// A function block containing multiple file handling methods. 
// Note that the body of this FB does NOT need to be called as it holds no logic.
// All the methods should be called untill they return true, if they provide error information, 
// it will be trough a reference variable.
//
// For examples refer to tests in the folder "TESTS/Test suites", file "FB_FileHandlerTests".

{attribute 'no_explicit_call' := 'Body contains no logic, calling methods only allowed.'}
FUNCTION_BLOCK FB_FileHandler EXTENDS ZigaLibs_Core.FB_ErrorSource IMPLEMENTS I_FileHandler

VAR
	_fileInfo		: ST_FileInfo;
	_netId			: Tc2_System.T_AmsNetID;
	_lastOpenMode	: E_FileOpenMode;
	_streamEmpty	: BOOL := TRUE;
END_VAR

// Closes the file and returns TRUE when done.
METHOD Close : BOOL
Close := THIS^.CloseSilent(FALSE);
END_METHOD

// Closes the file without clearing the file properties.
METHOD PRIVATE CloseSilent : BOOL
VAR_INPUT
	silent	: BOOL; // IF set to TRUE, the file property won't be modified. To be used when flushing the stream.
END_VAR
VAR_INST
	fbFileClose	: Tc2_System.FB_FileClose;
END_VAR

VAR
	varInfo	: ZigaLibs_Core.T_VarInfo;
END_VAR
fbFileClose(
	bExecute := NOT fbFileClose.bBusy,
	hFile := File.Handle,
	sNetId := File.NetId);

IF NOT fbFileClose.bBusy THEN
	CloseSilent := TRUE;
	IF fbFileClose.bError THEN
		varInfo := __VARINFO(fbFileClose);
		THIS^.RaiseAdsError(Tc2_Standard.CONCAT(THIS^.InstancePath, varInfo.Symbol), fbFileClose.nErrId);
		THIS^.GenericError.Message := Tc2_Standard.CONCAT('An error occured when closing the file ', File.Name);
		fbFileClose(bExecute := FALSE);	
		RETURN;
	END_IF
	
	_streamEmpty := TRUE;
	fbFileClose(bExecute := FALSE);
	File.Handle := 0;	
	IF NOT silent THEN
		File.IsOpened := FALSE;
	END_IF
END_IF
END_METHOD

// Creates the file, if it does not yet exist,
METHOD Create : BOOL
VAR_INPUT
	path	: Tc2_System.T_MaxString;	// Path to the file location
	name	: Tc2_System.T_MaxString;	// Name of the file
	netId	: Tc2_System.T_AmsNetID;	// NetId where the file is located
END_VAR
VAR
	sb	: ZigaLibs_Core.FB_StringBuilder;
END_VAR
IF NOT file.IsOpened THEN
	THIS^.Open(
		path := path,
		name := name,
		mode := E_FileOpenMode.BINARY_APPEND_OVERWRITE_EXISTING,
		netId := netId);
		
	// Error opening the file, report and stop.
	IF THIS^.Error THEN
		THIS^.GenericError.Source := sb.Reset()
			.AddString(THIS^.InstancePath)
			.AddString('.Create()')
			.Create();
		
		THIS^.GenericError.Message := sb.Reset()
			.AddString('An error occurred when creating the file, while opening it:')
			.AddString(' Path = ').AddWithDblQuotationMarks(path)
			.AddString(' Name = ').AddWithDblQuotationMarks(name)
			.AddString(' NetId = ').AddWithDblQuotationMarks(netId)
			.AddString('. Refer to AdsError for more info.')
			.Create();
		Create := TRUE;
		RETURN;
	END_IF
ELSE
	Create := THIS^.Close();
	
	// Error closing the file. Report and stop.
	IF THIS^.Error THEN
		THIS^.GenericError.Source := sb.Reset()
			.AddString(THIS^.InstancePath)
			.AddString('.Create()')
			.Create();
		THIS^.GenericError.Message := sb.Reset()
			.AddString('An error occurred when creating the file, while closing it:')
			.AddString(' Path = ').AddWithDblQuotationMarks(path)
			.AddString(' Name = ').AddWithDblQuotationMarks(name)
			.AddString(' NetId = ').AddWithDblQuotationMarks(netId)
			.AddString('. Refer to AdsError for more info.')
			.Create();
	END_IF
END_IF
END_METHOD

{attribute 'monitoring':='call'}
(* Gets the current file properties.*)
PROPERTY File : REFERENCE TO ST_FileInfo
GET
File REF= _fileInfo;
END_GET
SET // PROTECTED
_fileInfo := File;
END_SET
END_PROPERTY

// Flushes the current file stream data to the file. 
// Basically file is closed and re-opened, which in turn writes the content of the stream to the file.
// If the file was opened to overwrite existing content, flushing will clear the data in the file!
// While flushing is being executed, the .File property DOES NOT CHANGE 
// For example, the File.IsOpened will remain TRUE even at the point where it is actually not. It will then be re-opened. 
// If an error occurs however, properties will be set to correct state.

METHOD Flush : BOOL
VAR_INST
	closeDone		: BOOL;
END_VAR
IF closeDone OR_ELSE THIS^.CloseSilent(TRUE) THEN
	// Error closing the file while flushing...
	IF THIS^.Error AND NOT closeDone THEN
		Flush := TRUE;
		THIS^.GenericError.Message := 'An error occurred while flushing the file stream (closing the file)...';
		THIS^.GenericError.Source := Tc2_Standard.CONCAT(THIS^.InstanceName, '.Flush()');
		RETURN;
	END_IF
	
	closeDone := TRUE;
END_IF

IF closeDone AND_THEN THIS^.Open(File.Path, File.Name, _lastOpenMode, File.NetId) THEN
	closeDone := FALSE;
	Flush := TRUE;
	// Error while opening the file while flushing...
	IF THIS^.Error THEN
		THIS^.File.Handle := 0;
		THIS^.File.IsOpened := FALSE;
		THIS^.GenericError.Message := 'An error occurred while flushing the file stream (opening the file)...';
		THIS^.GenericError.Source := Tc2_Standard.CONCAT(THIS^.InstanceName, '.Flush()');
	END_IF
END_IF
END_METHOD

// Opens the file in the path provided. If a file is already opened nothing happens.
// Returns: TRUE when done.
METHOD Open : BOOL
VAR_INPUT
	path	: Tc2_System.T_MaxString;	// Path to the file location
	name	: Tc2_System.T_MaxString;	// Name of the file
	mode	: E_FileOpenMode;			// Mode in which the file will be opened
	netId	: Tc2_System.T_AmsNetID;	// NetId where the file is located
END_VAR

VAR_INST
	fbFileOpen	: Tc2_System.FB_FileOpen;
END_VAR

VAR
	varInfo	: ZigaLibs_Core.T_VarInfo;
END_VAR
IF THIS^.File.Handle <> 0 THEN
	Open := TRUE;
	RETURN;
END_IF

fbFileOpen(
	bExecute := NOT fbFileOpen.bBusy,
	nMode := mode,
	sNetId := netID,
	sPathName := Utilities.Path.Generate().Join(path).Join(name).Create());
	
IF NOT fbFileOpen.bBusy THEN
	Open := TRUE;
	IF fbFileOpen.bError THEN
		varInfo := __VARINFO(fbFileOpen);
		THIS^.RaiseAdsError(Tc2_Standard.CONCAT(THIS^.InstancePath, varInfo.Symbol), fbFileOpen.nErrId);
		fbFileOpen(bExecute := FALSE);
		RETURN;
	END_IF
	_lastOpenMode := mode;
	fbFileOpen(bExecute := FALSE);
	File.Handle := fbFileOpen.hFile;
	File.Name := name;
	File.Path := path;
	File.NetId := netId;
	File.IsOpened := TRUE;
END_IF
END_METHOD

// Raise an error for a certain FB instance (calls from methods)
METHOD PROTECTED RaiseAdsError : BOOL
VAR_INPUT
	source	: STRING;
	code 	: UDINT;
END_VAR
THIS^.AdsError.Code := TcError.ToAdsErrorCode(code);
THIS^.AdsError.Source := source;
THIS^.Error := TRUE;
END_METHOD

// Reads the file and writes the content to the result variable.
// Returns TRUE when done.
METHOD Read : BOOL

VAR_INPUT
	result	: ANY;
END_VAR

VAR_INST
	fbFileRead	: Tc2_System.FB_FileRead;
	test	: Tc2_System.T_MaxString;
END_VAR

VAR
	varInfo	: ZigaLibs_Core.T_VarInfo;
END_VAR
fbFileRead(
	bExecute := NOT fbFileRead.bBusy,
	sNetId := File.NetId,
	hFile := File.Handle,
	pReadBuff := result.pValue,
	cbReadLen := DINT_TO_UDINT(result.diSize));
	
IF NOT fbFileRead.bBusy THEN
	Read := TRUE;
	IF fbFileRead.bError THEN
		varInfo := __VARINFO(fbFileRead);
		THIS^.GenericError.Message := Tc2_Standard.CONCAT('An error occured when reading the file ', File.Name);
		THIS^.RaiseAdsError(Tc2_Standard.CONCAT(THIS^.InstancePath, varInfo.Symbol), fbFileRead.nErrId);
		fbFileRead(bExecute := FALSE);
	END_IF
END_IF
END_METHOD

// Reset any existing error.
METHOD Reset
THIS^.ResetError();
END_METHOD

(* Returns TRUE if there is no content in the file stream.*)
{attribute'monitoring':='call'}
PROPERTY StreamEmpty : BOOL
GET
StreamEmpty := _streamEmpty;
END_GET
END_PROPERTY

// Writes binary content to the file.
// Returns TRUE when done.
METHOD WriteBinary : BOOL

VAR_INPUT
	data		: ANY;	// Bincary content to be written
END_VAR

VAR_INST
	fbFileWrite		: Tc2_System.FB_FileWrite;
END_VAR
VAR
	varInfo	: ZigaLibs_Core.T_VarInfo;
END_VAR
_streamEmpty := FALSE;

fbFileWrite(
	bExecute := NOT fbFileWrite.bBusy,
	sNetId := File.NetId,
	hFile := File.Handle,
	pWriteBuff := data.pValue,
	cbWriteLen := DINT_TO_UDINT(data.diSize));
	
IF NOT fbFileWrite.bBusy THEN
	IF fbFileWrite.bError THEN
		varInfo := __VARINFO(fbFileWrite);
		THIS^.RaiseAdsError(Tc2_Standard.CONCAT(THIS^.InstancePath, varInfo.Symbol), fbFileWrite.nErrId);
		WriteBinary := TRUE;
		fbFileWrite(bExecute := FALSE);
		RETURN;
	END_IF
	WriteBinary := TRUE;
	fbFileWrite(bExecute := FALSE);
	_streamEmpty := FALSE;
END_IF
END_METHOD

// Writes a single line to the file
// Returns TRUE when done.
METHOD WriteLine : BOOL

VAR_INPUT
	line : Tc2_System.T_MaxString;	// Text to be written
END_VAR

VAR_INST
	fbFilePuts 		: Tc2_System.FB_FilePuts;
END_VAR

VAR
	varInfo	: ZigaLibs_Core.T_VarInfo;
END_VAR
fbFilePuts(
	bExecute := NOT fbFilePuts.bBusy,
	sNetId := File.NetId,
	hFile := File.Handle,
	sLine := line);
	
IF NOT fbFilePuts.bBusy THEN
	IF fbFilePuts.bError THEN
		varInfo := __VARINFO(fbFilePuts);
		THIS^.RaiseAdsError(Tc2_Standard.CONCAT(THIS^.InstancePath, varInfo.Symbol), fbFilePuts.nErrId);
		fbFilePuts(bExecute := FALSE);
		WriteLine := TRUE;
		RETURN;
	END_IF
	_streamEmpty := FALSE;
	WriteLine := TRUE;
	fbFilePuts(bExecute := FALSE);
END_IF
END_METHOD

END_FUNCTION_BLOCK

(* stored: Version 1.1.0.1, ProductVersion 3.1.4024.14
   POU FB_FileHandler: Id {ced76f9f-82d7-00ef-2259-233acd438959}, SpecialFunc None
   Method Close: Id {fd83d39e-5189-0d8d-30a1-fc0cd272c0e3}
   Method CloseSilent: Id {e1d20dca-b669-0865-11b7-99db0287f0f9}
   Method Create: Id {db135558-7082-0976-0533-068312031e70}
   Property File: Id {af587ba4-f1af-0723-10cc-2475f9362808}
   Get Get: Id {a5cf36d4-84c2-0626-0d42-bfe92224b35a}
   Set Set: Id {7f2a75a3-5c5e-009d-2e8b-0623e7b1209f}
   Method Flush: Id {348ffd5a-b3da-06ae-2382-55605fe66f35}
   Method Open: Id {7d720987-37e9-0fce-1fc8-b172b6327f39}
   Method RaiseAdsError: Id {11bb7eac-00b2-0545-18dd-8c65e0bb7ac7}
   Method Read: Id {f0e75126-46de-08dd-11f7-1487dff764b1}
   Method Reset: Id {46d8a829-a30e-06ac-3c2a-ff8223a84623}
   Property StreamEmpty: Id {cd56f0e7-bde1-07db-06d6-50ba8347cba7}
   Get Get: Id {b10d77ee-ab6d-0005-3f06-9ac99420dd4c}
   Method WriteBinary: Id {dec0a7b1-f937-092c-23b6-95753861b16f}
   Method WriteLine: Id {27555d66-493b-0776-001f-cf9f50c82f71} *)
